(* CoDeSys 2.3 export: NETVARUDPDIAGSTRUCT.EXP *)

(* Data type *)
TYPE NetVarUDPDiagStruct :
STRUCT
	nSendCount		: UDINT;
	tLastSend			: TIME;
	nReceiveCount	: UDINT;
	tLastReceive		: TIME;
	nWriteCount		: UDINT;
	sLastError			: NetVarUDPError;
	tLastError			: TIME;
	nErrorCount		: UINT;
	nAcknowledges	: UINT;
END_STRUCT
END_TYPE
